{attribute 'qualified_only'}
VAR_GLOBAL CONSTANT
	ALARM_MAX_COUNT: UINT := 3;
END_VAR

(* stored: Version 1.1.0.1, ProductVersion 3.1.4024.15
   GVL AlarmEventParam: Id {81f4bccd-ade8-4820-bb41-36ccddd6eee3}, ParameterList True *)
